FUNCTION_BLOCK FB_MotorControlInverter EXTENDS FB_MotorControlReverse
VAR
	resetButton		: Button;	// Scada Button inverter reset
	speedEdit		: NumberEdit; // SCADA number Edit field
	currentSpeed	: REAL;	  // Current speed read from Inverter
	
	iDriveInverter  : I_DriveInverter; // interface variable
	
	
END_VAR

SUPER^(); //call base class 

IF resetButton.IsPressed THEN
	Reset();
END_IF

METHOD FB_init : BOOL
VAR_INPUT
	bInitRetains : BOOL; // if TRUE, the retain variables are initialized (warm start / cold start)
	bInCopyCode  : BOOL;  // if TRUE, the instance afterwards gets moved into the copy code (online change)
	iDrive		 : I_Drive;
			
END_VAR
//check it is possible conversion type of interface

IF __QUERYINTERFACE(iDrive, iDriveInverter) THEN
	bSuccess := TRUE;
END_IF
END_METHOD

METHOD Reset : BOOL
VAR_INPUT
END_VAR
iDriveInverter.Reset();
END_METHOD

METHOD Speed : BOOL
VAR_INPUT
	_setSpeedValue : REAL;
END_VAR
iDriveInverter.SetSpeed(_setSpeedValue);
END_METHOD

END_FUNCTION_BLOCK

(* stored: Version 1.1.0.1, ProductVersion 3.1.4024.12
   POU FB_MotorControlInverter: Id {09f97a7c-20ed-4dba-b4ed-2db01e0000dd}, SpecialFunc None
   Method FB_init: Id {0e59730c-83eb-413d-aa7a-18575dff9c7e}
   Method Reset: Id {021b8393-ba79-4dba-a194-82bb069c65c7}
   Method Speed: Id {e377fbfd-7497-4fa5-9059-0449f28386b6} *)
